// TIA Portal V17 export
// export: Created 2023-06-23T18:33:38.1093821Z, ExportSetting WithDefaults, DisplayName Totally Integrated Automation Portal, DisplayVersion V17, DisplayName TIA Portal Openness, DisplayVersion V17, DisplayName TIA Portal Version Control Interface, DisplayVersion V17, DisplayName STEP 7 Professional, DisplayVersion V17, DisplayName STEP 7 Safety, DisplayVersion V17, DisplayName WinCC Advanced / Unified PC, DisplayVersion V17
VAR_GLOBAL   // PLC tag table "07_CT-1"
   "iCT-1" AT %I1.4 : Bool;
   "oCT-1s" AT %Q20.2 : Bool;
   "oCT-1f" AT %Q20.3 : Bool;
END_VAR
